// TIA Portal V21 export
DATA_BLOCK "InterfaceDB"   // DB2
{ S7_Optimized_Access := 'TRUE' }
// stored: MemoryReserve 100
   VAR
      ksd1 : "coneCrusherIOs";
   END_VAR
BEGIN
END_DATA_BLOCK
